Staubli VAL3: onStart.pgx

program onStart()
  local num l_nSize
  local frame l_fNewWorld
begin
  // load the default gun
  if !cycleStatus:bCycle
    call tcp:getSize(l_nSize)
    if saveData:nIndexTool>=l_nSize
      // BAD GUN INDEX load default ZERO
      saveData:nIndexTool=0
    endIf
    // get the tool
    call tcp:getTool(saveData:tTool,saveData:nIndexTool)
    fFrame.trsf=saveData:fFrameItem[saveData:nFrameActive].fFrame.trsf
    $jogContext(saveData:tTool,fFrame,0)
  endIf
  //
  // logMsg
  logMsg("[KERNEL] INTERFACE:PAGE Advance")
  //
  use:bUseRefresh=true
end
